// TIA Portal V20 export
DATA_BLOCK "ModuleTypePackageRevision"   // DB99
TITLE = ModuleTypePackageRevision
{ S7_Optimized_Access := 'TRUE' }
AUTHOR : Siemens AG
FAMILY : MTP
VERSION : 1.0
// The version information of the entire MTP
// stored: InstanceOfName typeMTPModuleTypePackageRevision, InstanceOfType UDT
"typeMTPModuleTypePackageRevision"
   // VAR
   //    ModuleTypePackageRevision { ExternalAccessible := 'False'; ExternalVisible := 'False'; ExternalWritable := 'False'} : String := '3.0.0';
   // END_VAR
BEGIN
END_DATA_BLOCK
